// TIA Portal V20 export
FUNCTION_BLOCK "FB_LaserAirProcess"   // FB432, SCL
{ S7_Optimized_Access := 'TRUE' }
// stored: AutoNumber false, MemoryReserve 100, SetENOAutomatically false
   VAR
      sTimeDelay : Time;
      sTimerGas : TON_TIME;
      sGasAssistOn : Bool;
      sLaser_Air_Process_Ctrl { S7_SetPoint := 'True'} : "FB_AnalogInputThreshold";
      sNozzle_Over_Pressure { S7_SetPoint := 'True'} : "FB_AnalogInputThreshold";
      sGasAssistDelay { ExternalAccessible := 'False'; ExternalVisible := 'False'; ExternalWritable := 'False'} : Bool;
      sGasAssistStartCh1 : Bool;
      sGasAssistStartCh2 : Bool;
      sGasAssistByKey : Bool;
      sGasReadValue : Bool;
      sRT_sGasAssistStartCh1 : R_TRIG;
      sRT_sGasAssistStartCh2 { S7_SetPoint := 'True'} : R_TRIG;
      sFT_sGasAssistStartCh1 { S7_SetPoint := 'True'} : F_TRIG;
      sFT_sGasAssistStartCh2 { S7_SetPoint := 'True'} : F_TRIG;
      sGasAssistSetPointJog { S7_SetPoint := 'True'} : Real;
      sGasAssistOffTimer : TOF_TIME;
   END_VAR
   VAR_TEMP
      tReadError : Bool;
      tErrorCode : Int;
   END_VAR
   VAR CONSTANT
      GAS_ASSIST_TIME : Time := T#5m;
   END_VAR
BEGIN
   REGION Description header 
       //==================================================================================
       // POSALUX Swiss SA / (C) Copyright 2024
       //----------------------------------------------------------------------------------
       // Title: Laser AirProcess
       // Comment/Function: 
       //
       // Author: Gowsigan SRITHARAN
       // Engineering: TIA Portal v17
       //----------------------------------------------------------------------------------
       // Change log table:
       // Version  | Date     | Expert in charge | Changes applied
       // ---------|----------|------------------|------------------------------------
       // 00.00.01 | 20241205 | GSR              | First released version
       // 00.00.02 | 20250314 | WFA              | Management modifications in Jog Mode
       // ==================================================================================
   END_REGION

   REGION Gas Assist ON
       "DB_DigitalOutputs".sGasAssistOn.sSWStatus := "DB_PowerOn".sMachineReadySoft;
   END_REGION

   REGION Disable Gas Assist Key[2]
       "DB_McpKeyboardSignals".sK2_GasAssist.sKeyDisable :=
       NOT "LBP_ModeGroup".E_JOG
       OR "LBP_Chan1".E_ProgRunning
       OR "LBP_Chan1".E_ProgStop
       OR "LBP_Chan1".E_ProgWait
       OR "DB_GestionWorkingModes".sMCP_KxxKeysDisable;

       "DB_HmiKeyboardSignals".sK2_GasAssist.sKeyDisable :=
       NOT "LBP_ModeGroup".E_JOG
       OR "LBP_Chan1".E_ProgRunning
       OR "LBP_Chan1".E_ProgStop
       OR "LBP_Chan1".E_ProgWait;
   END_REGION

   REGION Gas Assist
       IF "LBP_Chan1".MDyn[90] THEN                                // M90 : Start Gas Assist
           #sGasAssistStartCh1 := TRUE;
       ELSIF "LBP_Chan1".MDyn[91] OR "LBP_Chan1".A_Reset THEN      // M91 : Stop Gas Assist
           #sGasAssistStartCh1 := FALSE;
       END_IF;
   END_REGION

   REGION Gas Assist by Key
       IF "DB_McpKeyboardSignals".sK2_GasAssist.sKeySWTogglePositiveFront
           OR "DB_HmiKeyboardSignals".sK2_GasAssist.sKeySWTogglePositiveFront THEN
           #sGasAssistByKey := TRUE;
       ELSIF "DB_McpKeyboardSignals".sK2_GasAssist.sKeySWToggleNegativeFront
           OR "DB_HmiKeyboardSignals".sK2_GasAssist.sKeySWToggleNegativeFront THEN
           #sGasAssistByKey := FALSE;
       END_IF;
   END_REGION

   REGION Gas Read Value
       #sRT_sGasAssistStartCh1(CLK := #sGasAssistStartCh1);
       #sFT_sGasAssistStartCh1(CLK := #sGasAssistStartCh1);

       IF #sRT_sGasAssistStartCh1.Q
           OR #sFT_sGasAssistStartCh1.Q THEN
               #sGasReadValue := TRUE;
       END_IF;
   END_REGION

   REGION Nitrogen Gas LED[2]
       "DB_McpKeyboardSignals".sK2_GasAssist.sLedSWStatus :=
       #sGasAssistStartCh1
       OR #sGasAssistByKey;

       "DB_HmiKeyboardSignals".sK2_GasAssist.sLedSWStatus :=
       #sGasAssistStartCh1
       OR #sGasAssistByKey;
   END_REGION

   REGION Laser Air Pressure Process Set Point
       "DB_DigitalOutputs".sLaserAirPressureProcess.sSWStatus :=
       #sGasAssistStartCh1
       OR #sGasAssistByKey;
   END_REGION

   REGION Gas Assist Set point
       "LBP_TransferSelData"(Enable := #sGasReadValue,
                             Funct := 16#03,
                             IVAR1 := 972,
                             IVAR2 := -1,
                             Error => #tReadError,
                             ErrCode => #tErrorCode,
                             S7Var := "DB_HMISetting".GasAssistSetPoint);

       // Gas Assist Set Point if Jog mode
       IF NOT "LBP_ModeGroup".E_JOG AND "DB_HMISetting".GasAssistSetPoint <> 0 AND #sGasReadValue THEN
           #sGasAssistSetPointJog := "DB_HMISetting".GasAssistSetPoint;
       ELSE
           #sGasAssistSetPointJog := "DB_Parameters".GazPressureManual;
        END_IF;   

       // Transfer Gas Assist Set Point
        IF #sGasReadValue THEN
           IF "LBP_ModeGroup".E_JOG THEN
               "DB_AnalogInputDataHMI".Laser_Air_Pressure_Process.TargetValue := #sGasAssistSetPointJog;
               "DB_AnalogInputDataHMI".Nozzle_Overpressure.TargetValue := #sGasAssistSetPointJog;
           ELSE
               "DB_AnalogInputDataHMI".Laser_Air_Pressure_Process.TargetValue := "DB_HMISetting".GasAssistSetPoint;
               "DB_AnalogInputDataHMI".Nozzle_Overpressure.TargetValue := "DB_HMISetting".GasAssistSetPoint;
           END_IF;
       END_IF;

       // Reset Gas Assist Value by push Reset Button or after 5min no process
       #sGasAssistOffTimer(IN := ("LBP_Chan1".E_ProgRunning AND "LBP_Chan1".E_ProgRunning)
                           OR ("LBP_ModeGroup".E_JOG AND "DB_McpKeyboardSignals".sK2_GasAssist.sKeySWToggleStatus)
                           OR ("LBP_ModeGroup".E_JOG AND "DB_HmiKeyboardSignals".sK2_GasAssist.sKeySWToggleStatus),
                           PT := #GAS_ASSIST_TIME);

       // IF "MCP1_In".reset OR NOT #sGasAssistOffTimer.Q THEN
           IF "MCP1_In".reset THEN // WFA A REVOIR
           "DB_HMISetting".GasAssistSetPoint := 0.0;
           "DB_AnalogInputDataHMI".Laser_Air_Pressure_Process.TargetValue := 0.0;
           "DB_AnalogInputDataHMI".Nozzle_Overpressure.TargetValue := 0.0;
       END_IF;

       // Gas assist transfer to analog output
       IF NOT "LBP_ModeGroup".E_JOG THEN
           "DB_AnalogOutputs".sNozzleOverpressureSetPoint.sSWRealValue := "DB_HMISetting".GasAssistSetPoint;
       ELSE
           "DB_AnalogOutputs".sNozzleOverpressureSetPoint.sSWRealValue := #sGasAssistSetPointJog;
       END_IF;
   END_REGION

   REGION Laser Air process control
       #sLaser_Air_Process_Ctrl(iActualValue := "DB_AnalogInputs".sLaserAirPressureProcess.sSWRealValue,
                                iStartDelay := "DB_DigitalOutputs".sLaserAirPressureProcess.sSWStatus,
                                ioAlarmMin := "LBP_AlarmMsgs".UserA[06].A70UUxx[50],
                                ioWarningMin := "LBP_AlarmMsgs".UserA[07].A70UUxx[50],
                                ioWarningMax := "LBP_AlarmMsgs".UserA[07].A70UUxx[51],
                                ioAlarmMax := "LBP_AlarmMsgs".UserA[06].A70UUxx[51],
                                oDataAction => "DB_AnalogInputAction".Laser_Air_Pressure_Process,
                                iDataPLC := "DB_AnalogInputDataPLC".Laser_Air_Pressure_Process,
                                iDataHMI := "DB_AnalogInputDataHMI".Laser_Air_Pressure_Process);
     END_REGION

     REGION Regulation gas assist control
         #sNozzle_Over_Pressure(iActualValue := "DB_AnalogInputs".sNozzleOverpressure.sSWRealValue,
                                iStartDelay := "DB_DigitalOutputs".sLaserAirPressureProcess.sSWStatus,
                                ioAlarmMin := "LBP_AlarmMsgs".UserA[06].A70UUxx[60],
                                ioWarningMin := "LBP_AlarmMsgs".UserA[07].A70UUxx[60],
                                ioWarningMax := "LBP_AlarmMsgs".UserA[07].A70UUxx[61],
                                ioAlarmMax := "LBP_AlarmMsgs".UserA[06].A70UUxx[61],
                                oDataAction => "DB_AnalogInputAction".Nozzle_Overpressure,
                                iDataPLC := "DB_AnalogInputDataPLC".Nozzle_Overpressure,
                                iDataHMI := "DB_AnalogInputDataHMI".Nozzle_Overpressure);
     END_REGION
END_FUNCTION_BLOCK
